Staubli VAL3: compare.pgx

public program compare(num& x_nInput[], string x_sSign, num x_nCompareTo, bool& x_bResult[])
  local num l_nLength
  local num l_nElement
begin

  l_nLength = size(x_nInput)
  x_bResult[0] = false
  resize(x_bResult,1,l_nLength)

  switch x_sSign
    case ">"
      for l_nElement = 0 to l_nLength-1
        if x_nInput[l_nElement] > x_nCompareTo
          x_bResult[l_nElement] = true
        else
          x_bResult[l_nElement] = false
        endIf
      endFor
    break
    case ">="
      for l_nElement = 0 to l_nLength-1
        if x_nInput[l_nElement] >= x_nCompareTo
          x_bResult[l_nElement] = true
        else
          x_bResult[l_nElement] = false
        endIf
      endFor
    break
    case "<"
      for l_nElement = 0 to l_nLength-1
        if x_nInput[l_nElement] < x_nCompareTo
          x_bResult[l_nElement] = true
        else
          x_bResult[l_nElement] = false
        endIf
      endFor
    break
    case "<="
      for l_nElement = 0 to l_nLength-1
        if x_nInput[l_nElement] <= x_nCompareTo
          x_bResult[l_nElement] = true
        else
          x_bResult[l_nElement] = false
        endIf
      endFor
    break
    case "=="
      for l_nElement = 0 to l_nLength-1
        if x_nInput[l_nElement] == x_nCompareTo
          x_bResult[l_nElement] = true
        else
          x_bResult[l_nElement] = false
        endIf
      endFor
    break
  endSwitch
end
